% RSLogix 500 project I2P JOB 14_RUSSELL_BAK010.RSS, saved by version 10.00.00.00 %
PROJECT "ML02A"    % processor: Bul.1763 MicroLogix 1100 Series B %

PROGRAM FILES
  LAD 2   11 rungs

DATA FILES
  O0 OUTPUT  4 elements
  I1 INPUT  6 elements
  S2 STATUS  66 elements
  B3 BINARY  1 elements
  T4 TIMER  2 elements
  C5 COUNTER  1 elements
  R6 CONTROL  1 elements
  N7 INTEGER  1 elements
  F8 FLOAT  1 elements

LADDER 2
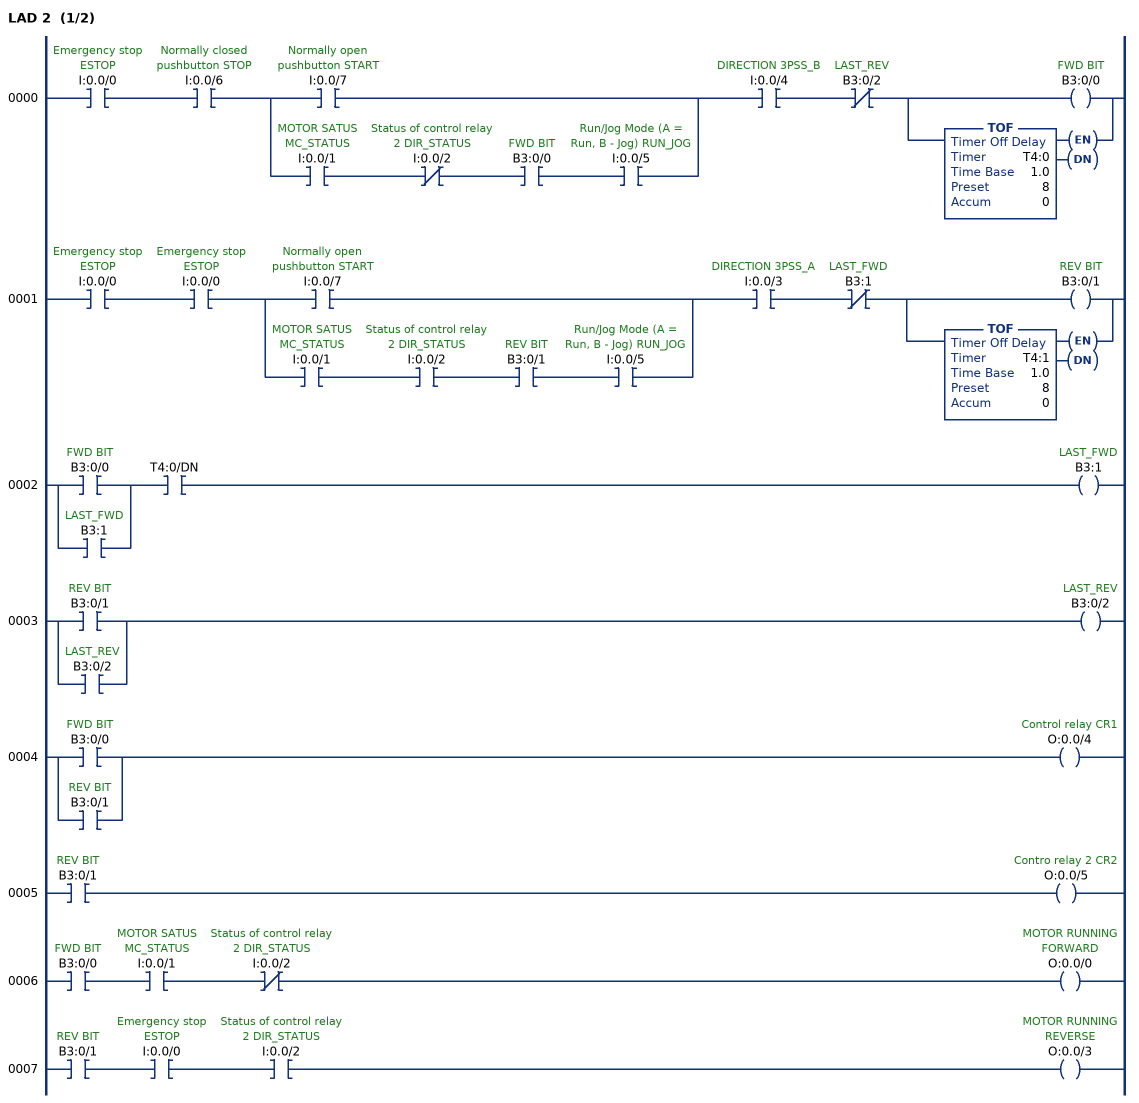
% Rung: 0 %
SOR XIC I:0.0/0 XIC I:0.0/6 BST XIC I:0.0/7 NXB XIC I:0.0/1 XIO I:0.0/2 XIC B3:0/0 XIC I:0.0/5 BND XIC I:0.0/4 XIO B3:0/2 BST OTE B3:0/0 NXB TOF T4:0 1.0 8 0 BND EOR
%   I:0.0/0  ESTOP  "Emergency stop" %
%   I:0.0/6  STOP  "Normally closed pushbutton" %
%   I:0.0/7  START  "Normally open pushbutton" %
%   I:0.0/1  MC_STATUS  "MOTOR SATUS" %
%   I:0.0/2  DIR_STATUS  "Status of control relay 2" %
%   B3:0/0  "FWD BIT" %
%   I:0.0/5  RUN_JOG  "Run/Jog Mode (A = Run, B - Jog)" %
%   I:0.0/4  3PSS_B  "DIRECTION" %
%   B3:0/2  LAST_REV %
% Rung: 1 %  % edit flag set %
SOR XIC I:0.0/0 XIC I:0.0/0 BST XIC I:0.0/7 NXB XIC I:0.0/1 XIC I:0.0/2 XIC B3:0/1 XIC I:0.0/5 BND XIC I:0.0/3 XIO B3:1 BST OTE B3:0/1 NXB TOF T4:1 1.0 8 0 BND EOR
%   I:0.0/0  ESTOP  "Emergency stop" %
%   I:0.0/7  START  "Normally open pushbutton" %
%   I:0.0/1  MC_STATUS  "MOTOR SATUS" %
%   I:0.0/2  DIR_STATUS  "Status of control relay 2" %
%   B3:0/1  "REV BIT" %
%   I:0.0/5  RUN_JOG  "Run/Jog Mode (A = Run, B - Jog)" %
%   I:0.0/3  3PSS_A  "DIRECTION" %
%   B3:1  LAST_FWD %
% Rung: 2 %  % edit flag set %
SOR BST XIC B3:0/0 NXB XIC B3:1 BND XIC T4:0/DN OTE B3:1 EOR
%   B3:0/0  "FWD BIT" %
%   B3:1  LAST_FWD %
% Rung: 3 %
SOR BST XIC B3:0/1 NXB XIC B3:0/2 BND OTE B3:0/2 EOR
%   B3:0/1  "REV BIT" %
%   B3:0/2  LAST_REV %
% Rung: 4 %
SOR BST XIC B3:0/0 NXB XIC B3:0/1 BND OTE O:0.0/4 EOR
%   B3:0/0  "FWD BIT" %
%   B3:0/1  "REV BIT" %
%   O:0.0/4  CR1  "Control relay" %
% Rung: 5 %
SOR XIC B3:0/1 OTE O:0.0/5 EOR
%   B3:0/1  "REV BIT" %
%   O:0.0/5  CR2  "Contro relay 2" %
% Rung: 6 %
SOR XIC B3:0/0 XIC I:0.0/1 XIO I:0.0/2 OTE O:0.0/0 EOR
%   B3:0/0  "FWD BIT" %
%   I:0.0/1  MC_STATUS  "MOTOR SATUS" %
%   I:0.0/2  DIR_STATUS  "Status of control relay 2" %
%   O:0.0/0  FORWARD  "MOTOR RUNNING" %
% Rung: 7 %
SOR XIC B3:0/1 XIC I:0.0/0 XIC I:0.0/2 OTE O:0.0/3 EOR
%   B3:0/1  "REV BIT" %
%   I:0.0/0  ESTOP  "Emergency stop" %
%   I:0.0/2  DIR_STATUS  "Status of control relay 2" %
%   O:0.0/3  REVERSE  "MOTOR RUNNING" %

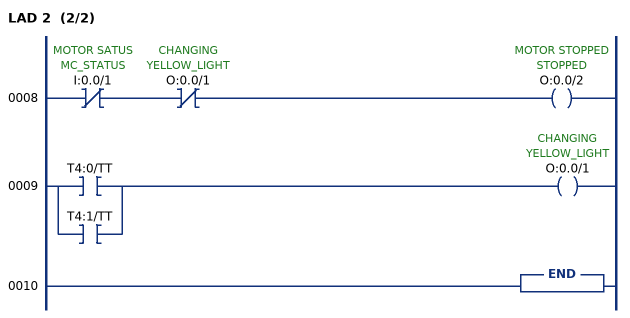
% Rung: 8 %  % edit flag set %
SOR XIO I:0.0/1 XIO O:0.0/1 OTE O:0.0/2 EOR
%   I:0.0/1  MC_STATUS  "MOTOR SATUS" %
%   O:0.0/1  YELLOW_LIGHT  "CHANGING" %
%   O:0.0/2  STOPPED  "MOTOR STOPPED" %
% Rung: 9 %
SOR BST XIC T4:0/TT NXB XIC T4:1/TT BND OTE O:0.0/1 EOR
%   O:0.0/1  YELLOW_LIGHT  "CHANGING" %
% Rung: 10 %
SOR END EOR

OTHER DOCUMENTED ADDRESSES
  I:0.0/8  JOG  "Normally open pushbutton"

COMMENTS NOT ATTACHED TO A CURRENT RUNG
  B3:0/0: Lucas Russell - JOB 12 - STOP-START-JOG using 3 pushbuttons for a 1p motor

DATA TABLE (non-zero values as saved)
DATA T4
% .PRE .ACC %
% T4:0 % 8 0
% T4:1 % 8 0
DATA C5
% .PRE .ACC %
% C5:0 % 16 8
